{attribute 'qualified_only'}
VAR_GLOBAL
		Device_1_EtherCAT : Device_1_EtherCAT_DC28AFF7;
END_VAR

(* stored: Version 1.2.0.0, ProductVersion 3.1.4024.9
   GVL GVL_iXlinker: Id {104633ef-c058-4fdd-bcef-0b0e50bce29b} *)
